(* IEC 61131-3 sources: JaccoSigma/tempclass/Class/FDD3000_VOVControl, 1 file *)

(* ---- FDD3000_VOVControl.st ---- *)
(*!
<Class
	Name               = "FDD3000_VOVControl"
	Revision           = "1.0"
	RealtimeTask       = "false"
	CyclicTask         = "false"
	BackgroundTask     = "false"
	Sigmatek           = "true"
	OSInterface        = "false"
	HighPriority       = "false"
	Automatic          = "false"
	UpdateMode         = "Prescan"
	SharedCommandTable = "true"
	Objectsize         = "(810,300)">
	<Channels>
		<Server Name="ActAutotuneStep" Visualized="true" Initialize="false" WriteProtected="false" Retentive="false" Comment="Shows the actual autotune step."/>
		<Server Name="ActCyclicStep" Visualized="true" Initialize="false" WriteProtected="false" Retentive="false" Comment="Shows actual cyclic step."/>
		<Server Name="ActLogData" Visualized="true" Initialize="false" WriteProtected="true" Retentive="false" Comment="Shows the amount of log entries."/>
		<Server Name="ActLSSStep" Visualized="true" Initialize="false" WriteProtected="false" Retentive="false" Comment="Shows the actual config step of node."/>
		<Server Name="ActSearchBitrate" Visualized="true" Initialize="false" WriteProtected="true" Retentive="false" Comment="Shows the actual search bitrate."/>
		<Server Name="ClassSvr" Visualized="false" Initialize="false" WriteProtected="true" Retentive="false" Comment="ClassSvr has no function."/>
		<Server Name="DataSource" Visualized="true" Initialize="false" WriteProtected="false" Retentive="false" Comment="Select data source to set / store parameters&#13;&#10;0 .. nothing select&#13;&#10;1 .. data from hardwareclass servers&#13;&#10;2 .. data actual on drive&#13;&#10;3 .. old data"/>
		<Server Name="FileSelect" Visualized="true" Initialize="false" WriteProtected="false" Retentive="false" Comment="Select if file with serial number or general file should be used.&#13;&#10;1 .. file with serial number (FDD3000_xxxxxxx.xml)&#13;&#10;2 .. file with general tag (FDD3000_General.xml)"/>
		<Server Name="MaxSpeed" Visualized="true" Initialize="false" WriteProtected="false" Retentive="false" Comment="Shows the maximum Speed of motor as rpm according to Motor Rated Frequency."/>
		<Server Name="MinSpeed" Visualized="true" Initialize="false" WriteProtected="false" Retentive="false" Comment="Shows the minimum Speed of motor as rpm according to Motor Rated Frequency."/>
		<Server Name="SetBitrate" Visualized="true" Initialize="false" WriteProtected="true" Retentive="false" Comment="Shows the bitrate of _CanOpenMng."/>
		<Server Name="SetDriveMode" Visualized="true" Initialize="false" WriteProtected="false" Retentive="false" Comment="Is used to set the Operation Mode of Drive if OpenLoop/RFC-A handling is started.&#13;&#10;1 .. Openloop&#13;&#10;2 .. RFC-A"/>
		<Server Name="SetNodeID" Visualized="true" Initialize="false" WriteProtected="true" Retentive="false" Comment="Shows the NodeID of the CanOpen Object."/>
		<Server Name="SetUserMotorParas" Visualized="true" Initialize="false" WriteProtected="false" Retentive="false" Comment="SetUserMotorParas is used to control steps at VOV.&#13;&#10;Autotune:&#13;&#10; 1 .. Start Autotune&#13;&#10;-1 .. Stop Autotune&#13;&#10;&#13;&#10;Openloop/RFC-A&#13;&#10;-1 .. Stop Openloop/RFC-A&#13;&#10;&#13;&#10;Drive Parameter&#13;&#10;11 .. Set Source Paras on HWK&#13;&#10;21 .. Load data from file&#13;&#10;22 .. Store data in file&#13;&#10;&#13;&#10;return values:&#13;&#10; 0 .. ok&#13;&#10;-1 .. failed to set source data on HWK Server &#13;&#10;-2 .. failed to load data from file&#13;&#10;-3 .. failed to store data in file"/>
		<Server Name="StartAutotune" Visualized="true" Initialize="false" WriteProtected="false" Retentive="false" Comment="Start Autotune Handling&#13;&#10;1 .. Start stationary Autotune&#13;&#10;2 .. Start rotating Autotune&#13;&#10;10 .. Start switch Operation Mode of Drive&#13;&#10;&#13;&#10;returncodes:&#13;&#10; 0 .. ok&#13;&#10;-1 .. Autotune failed&#13;&#10;-2 .. switch of Operation Mode failed"/>
		<Server Name="StartLSS" Visualized="true" Initialize="false" WriteProtected="false" Retentive="false" Comment="Is used to start configuring of node.&#13;&#10;1 .. start node config over LSS&#13;&#10;&#13;&#10;return value:&#13;&#10; 0 .. ok&#13;&#10;-1 .. node config failed."/>
		<Server Name="VOV_Active" Visualized="true" Initialize="false" WriteProtected="false" Retentive="false" Comment="Shows if VOV is active.&#13;&#10;0 .. not active&#13;&#10;1 .. active"/>
	</Channels>
	<Separators>
		<Servers>
			<SepChn Position="3"/>
			<SepChn Position="9"/>
			<SepChn Position="16"/>
			<SepChn Position="19"/>
		</Servers>
	</Separators>
	<RevDoku>
		<Owner Company="Sigmatek" Author="PieSte"/>
		<Dokumentation Revision="1.0" Date="02.02.2021" Author="ZoePat" Company="Sigmatek" Description="first library version"/>
	</RevDoku>
</Class>
*)
FDD3000_VOVControl : CLASS
	TYPE
	  eAutoTuneSSW :  //! <Type Public="true" Name="eAutoTuneSSW"/>
	  (
	    _IdleAutoTune,
	    _ReadActDriveMode,
	    _Wait4_ReadActDriveMode,
	    _Wait4InputDriveMode,
	    _SetDriveMode,
	    _Wait4SetDriveMode,
	    _StoreAndResetDrive,
	    _Wait4StoreAndResetDrive,
	    _NMTResetDrive,
	    _Wait4NMTResetDrive,
	    _Wait4ResetDrive,
	    _StoreOldParas,
	    _GetUserMotorParas,
	    _SetUserMotorParas,
	    _GetSTOState,
	    _InfoSTOEnable,
	    _SetAutoTuneDrive,
	    _Wait4_SetAutoTuneDrive,
	    _WarningAutoTuneStart,
	    _EnableAutoTune,
	    _Wait4AutoTuneFinished,
	    _Wait4Wait4AutoTuneFinished,
	    _GetAutoTuneParas,
	    _InfoSTODisable,
	    _DisableAutoTune,
	    _AutoTuneStopped,
	    _Wait4AutoTuneStopped,
	    _QuitErrorStopped,
	    _FinishedAutoTune,
	    _ErrorAutoTune
	  )$UDINT;
	  eCyclicSSW :  //! <Type Public="true" Name="eCyclicSSW"/>
	  (
	    _SDOCyclic,
	    _NodeSettings,
	    _AutoTune,
	    _SaveMotorParas,
	    _FileHandling
	  )$UDINT;
	  eLSSNodeSSW :  //! <Type Public="true" Name="eLSSNodeSSW"/>
	  (
	    _IdleLSS,
	    _DeactivateMng,
	    _SetLSSInfos,
	    _Wait4SetLSSInfos,
	    _WriteSDOCiA,
	    _StoreNodeConfig,
	    _Wait4StoreNodeConfig,
	    _ResetNode,
	    _Wait4ResetNode,
	    _ActivateMng,
	    _QuitErrorNode,
	    _FinishedLSS,
	    _ErrorLSS
	  )$UDINT;
	  eUserDriveMode :  //! <Type Public="true" Name="eUserDriveMode"/>
	  (
	    _ModeUnknown,
	    _OpenLoop,
	    _RFC_A
	  )$UDINT;
	  eUserMotorParas : DINT;
	END_TYPE
  //Servers:
	ClassSvr 	: SvrChCmd_DINT;
	VOV_Active 	: SvrCh_DINT;
	ActCyclicStep 	: SvrCh_eCyclicSSW_PTofCls_FDD3000_VOVControl;
	StartLSS 	: SvrCh_DINT;
	ActLSSStep 	: SvrCh_eLSSNodeSSW_PTofCls_FDD3000_VOVControl;
	SetNodeID 	: SvrCh_DINT;
	SetBitrate 	: SvrCh_DINT;
	ActSearchBitrate 	: SvrCh_DINT;
	StartAutotune 	: SvrCh_DINT;
	ActAutotuneStep 	: SvrCh_eAutoTuneSSW_PTofCls_FDD3000_VOVControl;
	SetDriveMode 	: SvrCh_eUserDriveMode_PTofCls_FDD3000_VOVControl;
	SetUserMotorParas 	: SvrCh_DINT;
	DataSource 	: SvrCh_DINT;
	FileSelect 	: SvrCh_DINT;
	MaxSpeed 	: SvrCh_DINT;
	MinSpeed 	: SvrCh_DINT;
	ActLogData 	: SvrCh_DINT;
  //Clients:
  //Variables:
  //Functions:

	FUNCTION VIRTUAL GLOBAL DataSource::Write
		VAR_INPUT
			input (EAX) 	: DINT;
		END_VAR
		VAR_OUTPUT
			result (EAX) 	: DINT;
		END_VAR;

	FUNCTION VIRTUAL GLOBAL FileSelect::Write
		VAR_INPUT
			input (EAX) 	: DINT;
		END_VAR
		VAR_OUTPUT
			result (EAX) 	: DINT;
		END_VAR;
  //Tables:
	FUNCTION @STD
		VAR_OUTPUT
			ret_code	: CONFSTATES;
		END_VAR;
	FUNCTION GLOBAL TAB @CT_;
END_CLASS;

FUNCTION VIRTUAL GLOBAL FDD3000_VOVControl::FileSelect::Write
	VAR_INPUT
		input (EAX) 	: DINT;
	END_VAR
	VAR_OUTPUT
		result (EAX) 	: DINT;
	END_VAR

  if input <> 2 then
    input := 1;
  else
    input := 2;
  end_if;

	FileSelect := input;
	result := FileSelect;

END_FUNCTION

FUNCTION VIRTUAL GLOBAL FDD3000_VOVControl::DataSource::Write
	VAR_INPUT
		input (EAX) 	: DINT;
	END_VAR
	VAR_OUTPUT
		result (EAX) 	: DINT;
	END_VAR

  if input < 0 | input > 4 then
    input := 0;
  end_if;

	DataSource := input;
	result := DataSource;

END_FUNCTION
